// SIMATIC STEP 7 (V5.x) project SortingByHeight
// CPU: CPU 314C-2 PN/DP
// station: P_ADR_BUS
// station: Hardware
// station: SIMATIC 300 Station

SYMBOL_TABLE
"SUPERVISOR_DB"	DB 1	FB 2
"R_TRIG"	FB 1	FB 1
"SUPERVISOR_FB"	FB 2	FB 2
"AT_ENTRY"	I 0.0	BOOL
"AT_FRONT"	I 0.1	BOOL
"LOW_BOX"	I 0.2	BOOL
"HIGH_BOX"	I 0.3	BOOL
"AT_UNLOAD_POS"	I 0.4	BOOL
"AT_RIGHT_EXIT"	I 0.5	BOOL
"AT_TURNABLE_ENTRY"	I 0.6	BOOL
"AT_LEFT_EXIT"	I 0.7	BOOL
"AT_LOAD_POS"	I 1.0	BOOL
"START"	I 1.1	BOOL
"TRIG1"	M 0.0	BOOL
"TRIG2"	M 0.1	BOOL
"TRIG3"	M 0.2	BOOL
"TRIG4"	M 0.3	BOOL
"TRIG5"	M 0.4	BOOL
"TRIG6"	M 0.5	BOOL
"TRIG7"	M 0.6	BOOL
"TRIG8"	M 0.7	BOOL
"TRIG9"	M 1.0	BOOL
"TRIG10"	M 1.1	BOOL
"TRIG11"	M 1.2	BOOL
"TRIG12"	M 1.3	BOOL
"TRIG13"	M 1.4	BOOL
"TRIG14"	M 1.5	BOOL
"LOW_BOX_TMP"	M 1.6	BOOL
"LOW_BOX_DETECTED"	M 1.7	BOOL
"HIGH_BOX_DETECTED"	M 2.0	BOOL
"AT_ENTRY_ACT1_E"	M 2.1	BOOL
"AT_ENTRY_ACT1_H"	M 2.2	BOOL
"AT_FRONT_ACT1_E"	M 2.3	BOOL
"AT_FRONT_ACT1_H"	M 2.4	BOOL
"AT_TURNABLE_ENTRY_ACT2_E"	M 2.5	BOOL
"AT_TURNABLE_ENTRY_ACT2_H"	M 2.6	BOOL
"AT_UNLOAD_POS_ACT_E"	M 2.7	BOOL
"AT_UNLOAD_POS_ACT_H"	M 3.0	BOOL
"AT_LEFT_EXIT_ACT2_E"	M 3.1	BOOL
"AT_LEFT_EXIT_ACT2_H"	M 3.2	BOOL
"AT_UNLOAD_POS_ACT2_E"	M 3.3	BOOL
"AT_UNLOAD_POS_ACT2_H"	M 3.4	BOOL
"AT_RIGHT_EXIT_ACT2_E"	M 3.5	BOOL
"AT_RIGHT_EXIT_ACT2_H"	M 3.6	BOOL
"VAR1"	M 3.7	BOOL
"VAR2"	M 4.0	BOOL
"VAR3"	M 4.1	BOOL
"VAR4"	M 4.2	BOOL
"LOW_BOX_DETECTED_E"	M 4.3	BOOL
"HIGH_BOX_DETECTED_E"	M 4.4	BOOL
"VAR5"	M 4.5	BOOL
"AT_TURNABLE_ENTRY_E"	M 4.6	BOOL
"AT_FRONT_ACT3_E"	M 4.7	BOOL
"AT_FRONT_ACT3_H"	M 5.0	BOOL
"TRIG15"	M 5.1	BOOL
"TRIG16"	M 5.2	BOOL
"TRIG17"	M 5.3	BOOL
"TRIG18"	M 5.4	BOOL
"TRIG19"	M 5.5	BOOL
"TRIG20"	M 5.6	BOOL
"HIGH_BOX_TMP"	M 5.7	BOOL
"TRIG21"	M 6.0	BOOL
"TRIG22"	M 6.1	BOOL
"START_E"	M 6.2	BOOL
"AT_TURNABLE_ENTRY_ACT1_E"	M 6.3	BOOL
"AT_TURNABLE_ENTRY_ACT1_H"	M 6.4	BOOL
"AT_FRONT_ACT2_E"	M 6.5	BOOL
"AT_FRONT_ACT2_H"	M 6.7	BOOL
"AT_UNLOAD_POS_ACT2_2_E"	M 7.0	BOOL
"AT_UNLOAD_POS_ACT2_2_H"	M 7.1	BOOL
"AT_TURNABLE_ENTRY_ACT3_E"	M 7.2	BOOL
"AT_TURNABLE_ENTRY_ACT3_H"	M 7.3	BOOL
"TRIG23"	M 7.4	BOOL
"TRIG24"	M 7.5	BOOL
"AT_TURNABLE_ENTRY_H"	M 7.6	BOOL
"TRIG25"	M 7.7	BOOL
"ENTRY_CONVEYOR_BUSY"	M 8.0	BOOL
"EMITTER"	Q 0.0	BOOL
"FEEDER_CONVEYOR"	Q 0.1	BOOL
"ENTRY_CONVEYOR"	Q 0.2	BOOL
"LOAD"	Q 0.3	BOOL
"TURN"	Q 0.4	BOOL
"LEFT_CONVEYOR"	Q 0.5	BOOL
"RIGHT_CONVEYOR"	Q 0.6	BOOL
"UNLOAD"	Q 0.7	BOOL
END_SYMBOL_TABLE

FUNCTION_BLOCK "R_TRIG"	// FB 1
VERSION : 0.0
VAR_INPUT
  CLK : BOOL ;
END_VAR
VAR_OUTPUT
  Q : BOOL ;
END_VAR
VAR
  SignalOld : BOOL ;
END_VAR
VAR_TEMP
  edge : BOOL ;
END_VAR
BEGIN
// body was compiled from an SCL source; compiled code not shown
END_FUNCTION_BLOCK

FUNCTION_BLOCK "SUPERVISOR_FB"	// FB 2
VERSION : 0.0
VAR_INPUT
  start_h : BOOL ;
  a_h : BOOL ;
  a_act_h : BOOL ;
  e_h : BOOL ;
  f_h : BOOL ;
  b_h : BOOL ;
  b_act_h : BOOL ;
  d_act_h : BOOL ;
  g_h : BOOL ;
  g_act2_2_h : BOOL ;
  d_h : BOOL ;
  g_act2_h : BOOL ;
END_VAR
VAR_OUTPUT
  start_e : BOOL ;
  a_e : BOOL ;
  a_act_e : BOOL ;
  e_e : BOOL ;
  f_e : BOOL ;
  b_e : BOOL ;
  b_act_e : BOOL ;
  d_act_e : BOOL ;
  g_e : BOOL ;
  g_act2_2_e : BOOL ;
  d_e : BOOL ;
  g_act2_e : BOOL ;
END_VAR
VAR
  start_t : FB 1;
  a_t : FB 1;
  a_act_t : FB 1;
  e_t : FB 1;
  f_t : FB 1;
  b_t : FB 1;
  b_act_t : FB 1;
  d_act_t : FB 1;
  g_t : FB 1;
  g_act2_2_t : FB 1;
  d_t : FB 1;
  g_act2_t : FB 1;
  continueSearch : BOOL  := TRUE;
  Q0_S0 : BOOL ;
  Q1_S0 : BOOL ;
  Q2_S0 : BOOL ;
  Q3_S0 : BOOL ;
  Q3_S1 : BOOL ;
  Q3_S7 : BOOL ;
  Q4_S2 : BOOL ;
  Q4_S8 : BOOL ;
  Q5_S10 : BOOL ;
  Q5_S11 : BOOL ;
  Q5_S12 : BOOL ;
  Q5_S3 : BOOL ;
  Q5_S4 : BOOL ;
  Q5_S5 : BOOL ;
  Q5_S6 : BOOL ;
  Q5_S9 : BOOL ;
  firstTime : BOOL  := TRUE;
END_VAR
BEGIN
// body was compiled from an SCL source; compiled code not shown
END_FUNCTION_BLOCK

DATA_BLOCK "SUPERVISOR_DB"	// DB 1
VERSION : 0.1
"SUPERVISOR_FB"
BEGIN
END_DATA_BLOCK

ORGANIZATION_BLOCK OB 1
TITLE = "Main Program Sweep (Cycle)"
VERSION : 0.1
VAR_TEMP
  OB1_EV_CLASS : BYTE ;	//Bits 0-3 = 1 (Coming event), Bits 4-7 = 1 (Event class 1)
  OB1_SCAN_1 : BYTE ;	//1 (Cold restart scan 1 of OB 1), 3 (Scan 2-n of OB 1)
  OB1_PRIORITY : BYTE ;	//Priority of OB Execution
  OB1_OB_NUMBR : BYTE ;	//1 (Organization block 1, OB1)
  OB1_RESERVED_1 : BYTE ;	//Reserved for system
  OB1_RESERVED_2 : BYTE ;	//Reserved for system
  OB1_PREV_CYCLE : INT ;	//Cycle time of previous OB1 scan (milliseconds)
  OB1_MIN_CYCLE : INT ;	//Minimum cycle time of OB1 (milliseconds)
  OB1_MAX_CYCLE : INT ;	//Maximum cycle time of OB1 (milliseconds)
  OB1_DATE_TIME : DATE_AND_TIME ;	//Date and time OB1 started
END_VAR
BEGIN
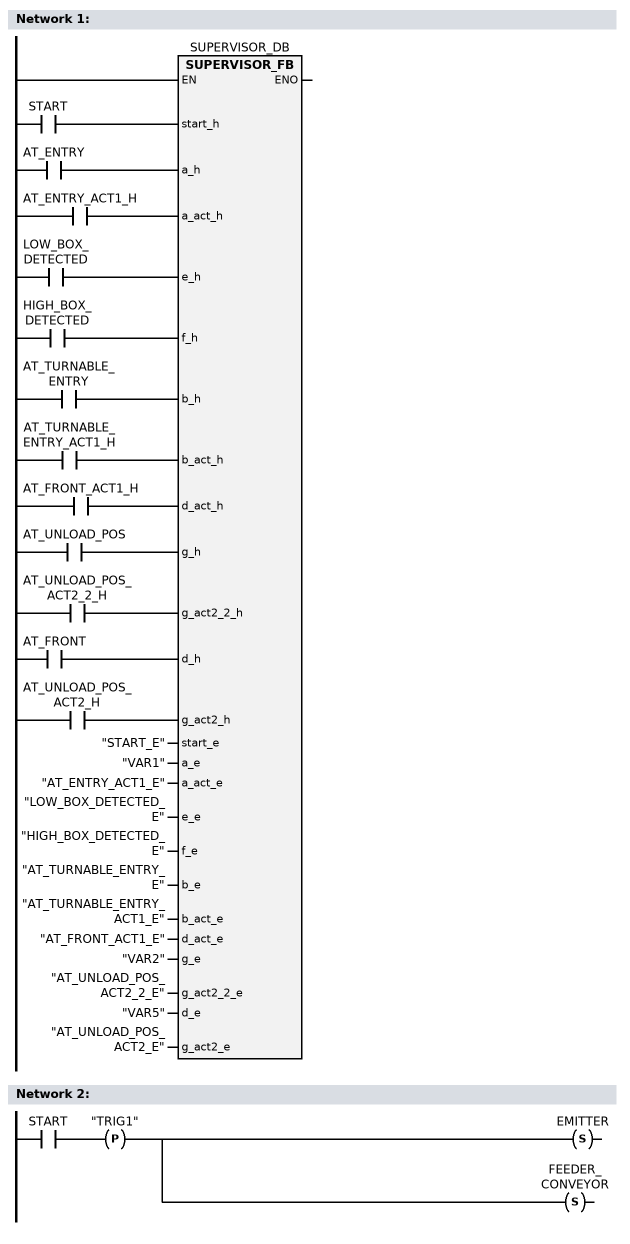
NETWORK
TITLE =
      A     "START";
      =     L 20.0;
      BLD   103;
      A     "AT_ENTRY";
      =     L 20.1;
      BLD   103;
      A     "AT_ENTRY_ACT1_H";
      =     L 20.2;
      BLD   103;
      A     "LOW_BOX_DETECTED";
      =     L 20.3;
      BLD   103;
      A     "HIGH_BOX_DETECTED";
      =     L 20.4;
      BLD   103;
      A     "AT_TURNABLE_ENTRY";
      =     L 20.5;
      BLD   103;
      A     "AT_TURNABLE_ENTRY_ACT1_H";
      =     L 20.6;
      BLD   103;
      A     "AT_FRONT_ACT1_H";
      =     L 20.7;
      BLD   103;
      A     "AT_UNLOAD_POS";
      =     L 21.0;
      BLD   103;
      A     "AT_UNLOAD_POS_ACT2_2_H";
      =     L 21.1;
      BLD   103;
      A     "AT_FRONT";
      =     L 21.2;
      BLD   103;
      A     "AT_UNLOAD_POS_ACT2_H";
      =     L 21.3;
      BLD   103;
      CALL  "SUPERVISOR_FB" , "SUPERVISOR_DB" (
           start_h                  := L 20.0,
           a_h                      := L 20.1,
           a_act_h                  := L 20.2,
           e_h                      := L 20.3,
           f_h                      := L 20.4,
           b_h                      := L 20.5,
           b_act_h                  := L 20.6,
           d_act_h                  := L 20.7,
           g_h                      := L 21.0,
           g_act2_2_h               := L 21.1,
           d_h                      := L 21.2,
           g_act2_h                 := L 21.3,
           start_e                  := "START_E",
           a_e                      := "VAR1",
           a_act_e                  := "AT_ENTRY_ACT1_E",
           e_e                      := "LOW_BOX_DETECTED_E",
           f_e                      := "HIGH_BOX_DETECTED_E",
           b_e                      := "AT_TURNABLE_ENTRY_E",
           b_act_e                  := "AT_TURNABLE_ENTRY_ACT1_E",
           d_act_e                  := "AT_FRONT_ACT1_E",
           g_e                      := "VAR2",
           g_act2_2_e               := "AT_UNLOAD_POS_ACT2_2_E",
           d_e                      := "VAR5",
           g_act2_e                 := "AT_UNLOAD_POS_ACT2_E");
      NOP   0;
NETWORK
TITLE =
      A     "START";
      FP    "TRIG1";
      S     "EMITTER";
      S     "FEEDER_CONVEYOR";
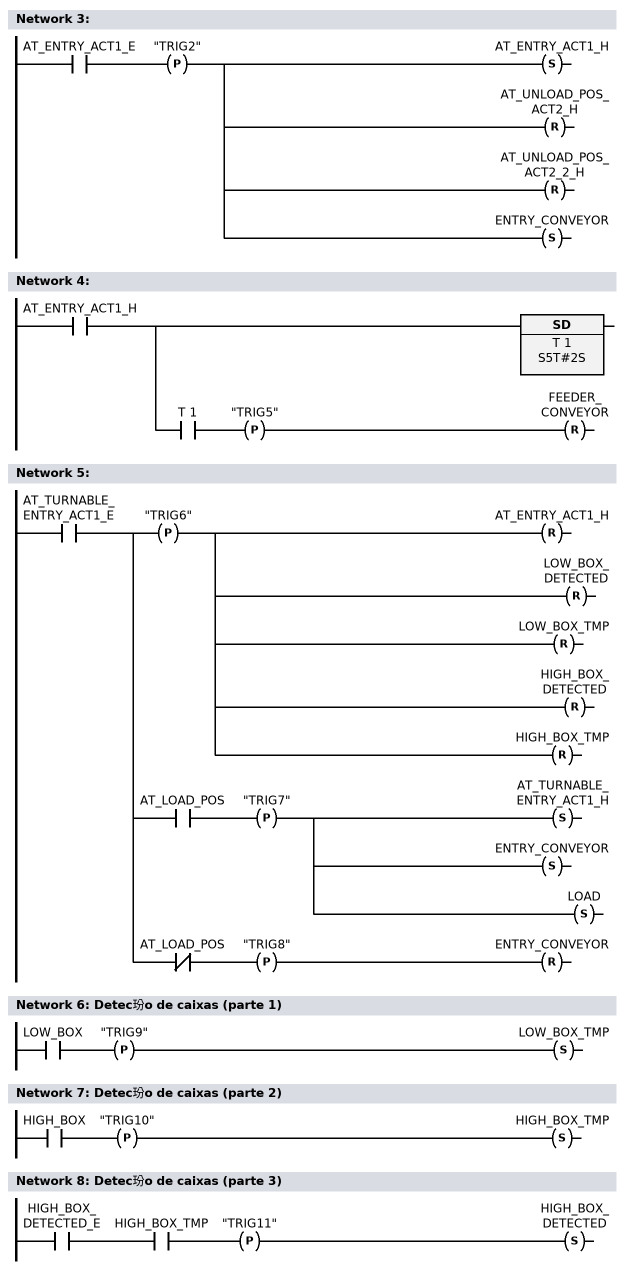
NETWORK
TITLE =
      A     "AT_ENTRY_ACT1_E";
      FP    "TRIG2";
      S     "AT_ENTRY_ACT1_H";
      R     "AT_UNLOAD_POS_ACT2_H";
      R     "AT_UNLOAD_POS_ACT2_2_H";
      S     "ENTRY_CONVEYOR";
NETWORK
TITLE =
      A     "AT_ENTRY_ACT1_H";
      =     L 20.0;
      A     L 20.0;
      BLD   102;
      L     S5T#2S;
      SD    T 1;
      A     L 20.0;
      A     T 1;
      FP    "TRIG5";
      R     "FEEDER_CONVEYOR";
NETWORK
TITLE =
      A     "AT_TURNABLE_ENTRY_ACT1_E";
      =     L 20.0;
      A     L 20.0;
      FP    "TRIG6";
      R     "AT_ENTRY_ACT1_H";
      R     "LOW_BOX_DETECTED";
      R     "LOW_BOX_TMP";
      R     "HIGH_BOX_DETECTED";
      R     "HIGH_BOX_TMP";
      A     L 20.0;
      A     "AT_LOAD_POS";
      FP    "TRIG7";
      S     "AT_TURNABLE_ENTRY_ACT1_H";
      S     "ENTRY_CONVEYOR";
      S     "LOAD";
      A     L 20.0;
      AN    "AT_LOAD_POS";
      FP    "TRIG8";
      R     "ENTRY_CONVEYOR";
NETWORK
TITLE = Detec玢o de caixas (parte 1)
      A     "LOW_BOX";
      FP    "TRIG9";
      S     "LOW_BOX_TMP";
NETWORK
TITLE = Detec玢o de caixas (parte 2)
      A     "HIGH_BOX";
      FP    "TRIG10";
      S     "HIGH_BOX_TMP";
NETWORK
TITLE = Detec玢o de caixas (parte 3)
      A     "HIGH_BOX_DETECTED_E";
      A     "HIGH_BOX_TMP";
      FP    "TRIG11";
      S     "HIGH_BOX_DETECTED";
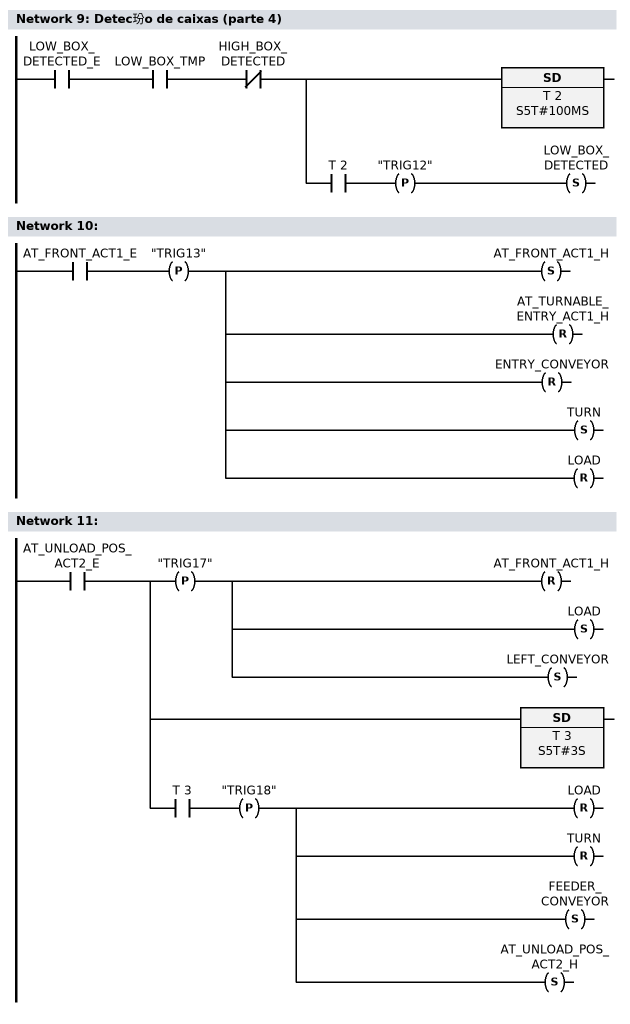
NETWORK
TITLE = Detec玢o de caixas (parte 4)
      A     "LOW_BOX_DETECTED_E";
      A     "LOW_BOX_TMP";
      AN    "HIGH_BOX_DETECTED";
      =     L 20.0;
      A     L 20.0;
      BLD   102;
      L     S5T#100MS;
      SD    T 2;
      A     L 20.0;
      A     T 2;
      FP    "TRIG12";
      S     "LOW_BOX_DETECTED";
NETWORK
TITLE =
      A     "AT_FRONT_ACT1_E";
      FP    "TRIG13";
      S     "AT_FRONT_ACT1_H";
      R     "AT_TURNABLE_ENTRY_ACT1_H";
      R     "ENTRY_CONVEYOR";
      S     "TURN";
      R     "LOAD";
NETWORK
TITLE =
      A     "AT_UNLOAD_POS_ACT2_E";
      =     L 20.0;
      A     L 20.0;
      FP    "TRIG17";
      R     "AT_FRONT_ACT1_H";
      S     "LOAD";
      S     "LEFT_CONVEYOR";
      A     L 20.0;
      BLD   102;
      L     S5T#3S;
      SD    T 3;
      A     L 20.0;
      A     T 3;
      FP    "TRIG18";
      R     "LOAD";
      R     "TURN";
      S     "FEEDER_CONVEYOR";
      S     "AT_UNLOAD_POS_ACT2_H";
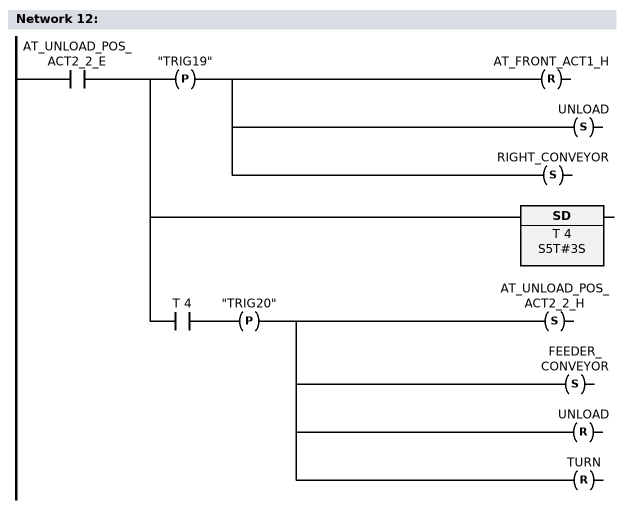
NETWORK
TITLE =
      A     "AT_UNLOAD_POS_ACT2_2_E";
      =     L 20.0;
      A     L 20.0;
      FP    "TRIG19";
      R     "AT_FRONT_ACT1_H";
      S     "UNLOAD";
      S     "RIGHT_CONVEYOR";
      A     L 20.0;
      BLD   102;
      L     S5T#3S;
      SD    T 4;
      A     L 20.0;
      A     T 4;
      FP    "TRIG20";
      S     "AT_UNLOAD_POS_ACT2_2_H";
      S     "FEEDER_CONVEYOR";
      R     "UNLOAD";
      R     "TURN";
END_ORGANIZATION_BLOCK
